// TIA Portal V19 export
FUNCTION "PosMatToPosAxis_Wheel" : LReal   // FC106, LAD
TITLE = From pos material to pos axis
// stored: Access Published, SetENOAutomatically false
   VAR_INPUT
      PosMaterial : LReal;
      Data : "MatCountData";
   END_VAR
   VAR_TEMP
      HalfModule : LReal;
      HalfNegativeModule : LReal;
      DeltaPosAx : LReal;
      DeltaMatCounter : LReal;
      AxPosCandidate : LReal;
   END_VAR
BEGIN

REGION Network 1: Half MODULE
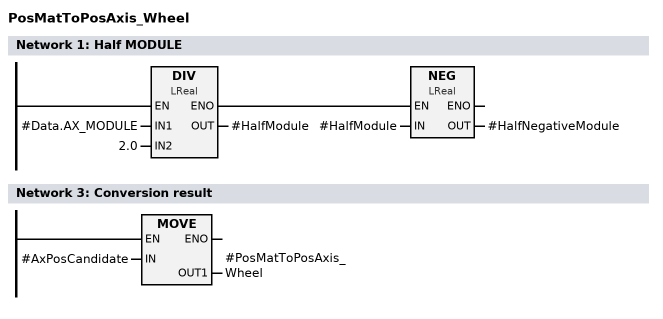
   RUNG wire#powerrail
      { S7_Templates := "SrcType := LReal" } Div(in1 := #Data.AX_MODULE, in2 := 2.0, out => #HalfModule)
      { S7_Templates := "SrcType := LReal" } Neg(in := #HalfModule, out => #HalfNegativeModule)
   END_RUNG
   // the same network as SCL:
   #HalfModule := #Data.AX_MODULE / 2.0;
   #HalfNegativeModule := -#HalfModule;
END_REGION

REGION Network 2 (SCL): Calculate position
   #DeltaMatCounter := #PosMaterial - #Data.CounterValue;

   IF #DeltaMatCounter > #HalfModule THEN
       #DeltaMatCounter := #DeltaMatCounter -#Data.AX_MODULE;
   ELSIF #DeltaMatCounter < #HalfNegativeModule THEN
       #DeltaMatCounter := #DeltaMatCounter + #Data.AX_MODULE;
   END_IF;

   #DeltaPosAx := #DeltaMatCounter;

   IF #Data.FAK > 0.0 THEN
       #DeltaPosAx := #DeltaMatCounter / #Data.FAK;
       #AxPosCandidate := #Data.AxPositionPrevious + #DeltaPosAx;
   END_IF;

   IF #AxPosCandidate > #Data.AX_MODULE THEN
       #AxPosCandidate := #AxPosCandidate - #Data.AX_MODULE;
   ELSIF #AxPosCandidate < 0.0 THEN
       #AxPosCandidate := #AxPosCandidate + #Data.AX_MODULE;
   END_IF;

   IF ABS_LREAL(#AxPosCandidate - #Data.AX_MODULE) < 0.01 THEN
       #AxPosCandidate := 0.0;
   END_IF;
END_REGION

REGION Network 3: Conversion result
   RUNG wire#powerrail
      Move(in := #AxPosCandidate, out1 => #PosMatToPosAxis_Wheel)
   END_RUNG
   // the same network as SCL:
   #PosMatToPosAxis_Wheel := #AxPosCandidate;
END_REGION
END_FUNCTION
